Staubli VAL3: J_goTo.pgx

program J_goTo(jointRx x_jPoint, num x_nIndex, bool& x_bUnreached[], string x_sName, num x_nMoveType, tool x_tTool)
  local bool l_bUnreached
  local num l_nIndexTool
  local tool l_tTool
  local num l_nMoveType
  local mdesc l_mDesc
begin
  // look for not cycle mode
  if !cycleStatus:bCycle
    if cycleStatus:nWorkingMode==1 and isPowered()
      // check for the index
      if nOldIndex!=x_nIndex or (cycleStatus:nWorkingStatus!=0 and cycleStatus:nWorkingStatus!=6)
        if !isEmpty()
          resetMotion()
        endIf
        if nOldIndex!=x_nIndex
          nOldIndex=x_nIndex
        endIf
      else
        if isEmpty() and cycleStatus:nWorkingStatus==0
          // get the data to move
          // use a sTemp mdesc to set the blend off
          l_mDesc.blend=off
          l_mDesc.accel=l_mDesc.decel=10
          l_mDesc.vel=10
          // use the got to of the trajectory...
          call J_MoveTo(x_jPoint,x_tTool,l_mDesc,x_nMoveType,x_bUnreached)
        endIf
      endIf
    else
      if cycleStatus:nWorkingMode!=1
        resetMotion()
      endIf
    endIf
  endIf
end
